PROGRAM Axis_10_Function_Blocks
VAR
END_VAR

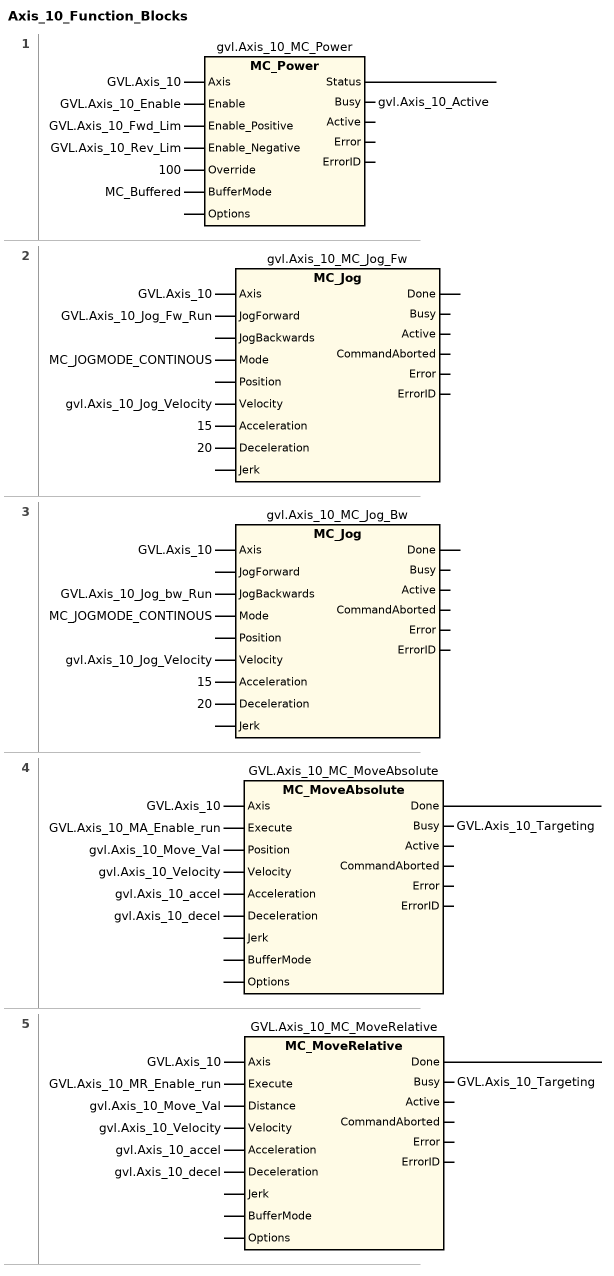
// NETWORK 1
gvl.Axis_10_MC_Power(
    Axis := GVL.Axis_10,
    Enable := GVL.Axis_10_Enable,
    Enable_Positive := GVL.Axis_10_Fwd_Lim,
    Enable_Negative := GVL.Axis_10_Rev_Lim,
    Override := 100,
    BufferMode := MC_Buffered,
    Busy => gvl.Axis_10_Active); // MC_Power

// NETWORK 2
gvl.Axis_10_MC_Jog_Fw(
    Axis := GVL.Axis_10,
    JogForward := GVL.Axis_10_Jog_Fw_Run,
    Mode := MC_JOGMODE_CONTINOUS,
    Velocity := gvl.Axis_10_Jog_Velocity,
    Acceleration := 15,
    Deceleration := 20); // MC_Jog

// NETWORK 3
gvl.Axis_10_MC_Jog_Bw(
    Axis := GVL.Axis_10,
    JogBackwards := GVL.Axis_10_Jog_bw_Run,
    Mode := MC_JOGMODE_CONTINOUS,
    Velocity := gvl.Axis_10_Jog_Velocity,
    Acceleration := 15,
    Deceleration := 20); // MC_Jog

// NETWORK 4
GVL.Axis_10_MC_MoveAbsolute(
    Axis := GVL.Axis_10,
    Execute := GVL.Axis_10_MA_Enable_run,
    Position := gvl.Axis_10_Move_Val,
    Velocity := gvl.Axis_10_Velocity,
    Acceleration := gvl.Axis_10_accel,
    Deceleration := gvl.Axis_10_decel,
    Busy => GVL.Axis_10_Targeting); // MC_MoveAbsolute

// NETWORK 5
GVL.Axis_10_MC_MoveRelative(
    Axis := GVL.Axis_10,
    Execute := GVL.Axis_10_MR_Enable_run,
    Distance := gvl.Axis_10_Move_Val,
    Velocity := gvl.Axis_10_Velocity,
    Acceleration := gvl.Axis_10_accel,
    Deceleration := gvl.Axis_10_decel,
    Busy => GVL.Axis_10_Targeting); // MC_MoveRelative

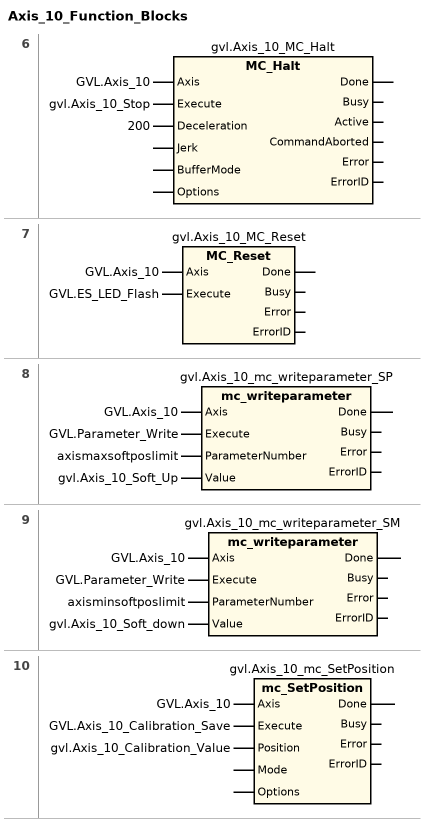
// NETWORK 6
gvl.Axis_10_MC_Halt(Axis := GVL.Axis_10, Execute := gvl.Axis_10_Stop, Deceleration := 200); // MC_Halt

// NETWORK 7
gvl.Axis_10_MC_Reset(Axis := GVL.Axis_10, Execute := GVL.ES_LED_Flash); // MC_Reset

// NETWORK 8
gvl.Axis_10_mc_writeparameter_SP(
    Axis := GVL.Axis_10,
    Execute := GVL.Parameter_Write,
    ParameterNumber := axismaxsoftposlimit,
    Value := gvl.Axis_10_Soft_Up); // mc_writeparameter

// NETWORK 9
gvl.Axis_10_mc_writeparameter_SM(
    Axis := GVL.Axis_10,
    Execute := GVL.Parameter_Write,
    ParameterNumber := axisminsoftposlimit,
    Value := gvl.Axis_10_Soft_down); // mc_writeparameter

// NETWORK 10
gvl.Axis_10_mc_SetPosition(
    Axis := GVL.Axis_10,
    Execute := GVL.Axis_10_Calibration_Save,
    Position := gvl.Axis_10_Calibration_Value); // mc_SetPosition

END_PROGRAM

(* stored: Version 1.1.0.1, ProductVersion 3.1.4022.12
   POU Axis_10_Function_Blocks: Id {b18dfb2a-0edf-4634-8eb8-1de04bdc4680}, SpecialFunc None *)
